(*======================================================================================================================================*)
(*fb_RS485Ping:	Einfacher Universal Ping Baustein um von allerlei Geräten von haus-bus.de Kommunikation zu Checken über RS485 
				im gegensatz zum ComCheck Baustein wird hier nur gelesen, da es Geräte gibt, welche entweder Zyklich selbst 
				ein Lebenszeichen geben z.B. CYD oder die 6Fach Taster (Helligkeit, Temp, Luftfeuchtigkeit).
				Besonderheit bei dem 6Fach Taster ist: nach einem Reset werden immer auch StatusTelegramme gesendet. 
				Damit lässt sich dann auch festellen ob ein Taster Online ist. 
				Für die Aktoren ist dieser Baustein eher weniger geeignet, da es dort keine Zyklischen Telegramme gibt und 
				auch nach einem Reset keine Statustelegramme gesendet werden! 
				
				Der Baustein kann auch verwendet werden um einfach nur zu überwachen, ob ein Teilnehmer noch online ist über langen
				Zeitraum- Dafür muss der Timeout einfach sehr Hoch gestellt werden - z.B 120 Minuten und bAutoPing Aktiviert sein 
			
				Wenn I_bAutoPing nicht Aktiv ist, wird nur eine Ping überprüfung beim Aktivieren des Bausteins über I_bExecute 
				durchgeführt. Wenn die Prüfung erfolgreich ist, wird der Status Q_bComOk gesetzt. Der Status Q_bComOk wird erst durch 
				I_bReset wieder zurück gesetzt. 
				
				Wenn I_bAutoPing Aktiv ist, wird sobald der Baustein über I_bExecute gestartet wurde, und ein Ping Aufgebaut ist, 
				immer nach ablauf der Zeit: I_tPingTimeout erneut der Ping geprüft. Sollte der Ping nicht kommen, so wird nach ablauf der 
+				Zeit: I_tPingTimeout in den Timepout gesprungen. Dann kann nur über einen Reset durch: I_bReset erneut gestartet werden*)
(*
Date          	| Version    	| created under        	| Author          	| Remark *)
(*====================================================================================================================================================*)
(*27/05/2025   	| 1.00      		| TC3		  		| N.Kersting       | first release *)
(*27/08/2025   	| 1.01      		| TC3		  		| N.Kersting       | Startup für Eventbaustein Implementiert *)
(*====================================================================================================================================================*)
FUNCTION_BLOCK fb_RS485Ping
VAR_INPUT
	I_bExecute			:BOOL;							(* Aktiviert den Ablauf *)
	I_bAutoPing			:BOOL;							(* Aktiviert die Automatische Prüfung, wenn aus- wird nur einmal beim Aktivieren über bExecute geprüft *)
	I_bAutoReset		:BOOL;							(* Aktiviert das Automatische wieder Quittieren wenn der Ping nicht empfangen wurde *)
	I_bReset			:BOOL;							(* Setzet den Ping und die Ablauf zurück *)
	I_tPingTimeout		:TIME := T#2S;					(* Zeit, bis der Ping gekommen sein muss *)
	I_diID				:DINT;							(* Device ID *)
	I_sStartZeichen		:BYTE := 16#FD;					(* Startzeichen Präfix *)
	I_sEndZeichen		:BYTE := 16#FE;					(* Endzeichen Suffix *)
	I_StringReceived	:STRING(255);					(* Empfangener String *)
END_VAR
VAR_OUTPUT		
	Q_sState			:STRING;						(* Status  *)
	Q_bComOk			:BOOL;							(* Verbindung Aufgebaut *)
	Q_bTimeout			:BOOL;							(* Timeout  *)
END_VAR
VAR
	bResetCnt			:BOOL;
	tonTimeout			:ton;
	icntSymbole			:INT;
	iStep				:INT;
	i					:INT;
	fbBusPingEvent		:fb_BusPingEvent;
	bCOMMem				:BOOL;
	rTrigFailCount		:r_trig;
	
	dwCntFail			:DWORD;
	bResetEvents		:BOOL := FALSE;
END_VAR

(* Timeout Zeit *)
tonTimeout(
	PT:= I_tPingTimeout);

(* Ping Fehler Zählen *)	
rTrigFailCount();
	
(* Reset ausführen *)
IF I_bReset 
	OR NOT I_bExecute
THEN
	iStep := 0;	
END_IF

(* Timeout Counter auf 0 Setzen *)
IF bResetCnt
THEN
	dwCntFail := 0;
END_IF
	
(* Ablauf *)
CASE iStep OF
(*=========================================================*)	
0:	Q_sState := 'INIT';
	Q_bComOk := FALSE;
	bResetEvents := FALSE;	(*Alle Events Reset ausführen *)
	bCOMMem := FALSE; (* Ping zurück setzen *)
	tonTimeout.IN := FALSE;
	Q_bTimeout := FALSE;
	rTrigFailCount.CLK := FALSE;
	
	IF I_bExecute
	THEN
		iStep := iStep +1;
	END_IF

(*============================================================================================*)	
1:	Q_sState := 'Setze alle Eventbausteine zurück';
	
	bResetEvents := TRUE;	(*Alle Events Reset ausführen *)

	IF NOT fbBusPingEvent.Q_bStartupDone 
	THEN
		iStep := iStep +1;
	END_IF
	
(*============================================================================================*)	
2:	Q_sState := 'Warte auf Startup Eventbausteine';
	
	bResetEvents := FALSE;	(*Alle Events Reset ausführen *)

	IF  fbBusPingEvent.Q_bStartupDone 
	THEN
		iStep := 10;
	END_IF	
	
(*=========================================================*)	
10:	Q_sState :=  'Warten auf Ping ';	
	tonTimeout.IN := TRUE;
	
	IF fbBusPingEvent.Q_bOut
	THEN
		tonTimeout.IN := FALSE;
		bCOMMem := TRUE;
		iStep := 998;
	ELSIF
		tonTimeout.Q
	THEN
		tonTimeout.IN := FALSE;
		Q_bTimeout := TRUE;
		Q_bComOk := FALSE;
		Q_sState :=  'Timeout- Kein Ping empfangen';	
		iStep := -1;
	END_IF

(*=========================================================*)	
998: Q_sState :=  'Ping empfangen, Warte das String Leer ist';	
	tonTimeout.IN := TRUE;
	
	IF NOT fbBusPingEvent.Q_bOut
	THEN
		iStep := 999;
	ELSIF
		tonTimeout.Q
	THEN
		tonTimeout.IN := FALSE;
		Q_bTimeout := TRUE;
		Q_bComOk := FALSE;
		Q_sState :=  'Timeout String wurde nicht geleert!';	
		iStep := -998;
	END_IF
	
(*=========================================================*)	
999: Q_sState :=  'Ping empfangen, erfolgreich Verbunden!';		
	Q_bComOk := TRUE;
	Q_bTimeout := FALSE;
	
	(* Die Verbindung wurde nun geprüft, kann aber nur über
		I_bReset wieder erneut geprüft werden ! *)
	
	IF I_bAutoPing
	THEN
		tonTimeout.IN := TRUE;
		
		IF tonTimeout.Q
		THEN
			tonTimeout.IN := FALSE;
				
			IF I_bExecute
			THEN
				iStep := 10;	(* Erneut Prüfen *)
			END_IF
		END_IF
	ELSE
		tonTimeout.IN := FALSE;
	END_IF
ELSE
(*=========================================================*)	
(*	Timeout *)	
	rTrigFailCount.CLK := TRUE;
	
	IF rTrigFailCount.Q
	THEN
		dwCntFail := dwCntFail+1;
	END_IF
	(*	Automatische Quittierung *)	
	IF 	I_bAutoReset
	THEN
		tonTimeout.IN := TRUE;
		
		IF tonTimeout.Q
			OR fbBusPingEvent.Q_bOut
		THEN
			tonTimeout.IN := FALSE;
			
			IF I_bExecute
			THEN
				rTrigFailCount.CLK := FALSE;
				iStep := 10;	(* Erneut Prüfen *)
			END_IF
		END_IF
	END_IF
END_CASE

(* Durchgehend Checken ob Ping kommt *)
fbBusPingEvent(
	I_bExecute :=			TRUE,
	I_bReset := 			bResetEvents,
	I_diID:= 				I_diID, 
	I_sReceivedString:= 	I_StringReceived, 
	Q_bOut=> 				);

END_FUNCTION_BLOCK

(* stored: Version 1.1.0.1, ProductVersion 3.1.4024.16
   POU fb_RS485Ping: Id {e37a6f29-62a1-4d1c-a02e-787c44742299}, SpecialFunc None *)
